{attribute 'linkalways'} 
{attribute 'no_explicit_call' := 'This FB is a CLASS and must be accessed using methods or properties'}
{attribute 'enable_dynamic_creation'}
FUNCTION_BLOCK FINAL EQ_LREAL EXTENDS Node
VAR
	in1 : _LREAL(0.0);
	in2 : _LREAL(0.0);
	out : _BOOL(FALSE);
END_VAR

METHOD PUBLIC Clone : I_Node
VAR
	pNode : POINTER TO EQ_LREAL;
END_VAR
pNode := __NEW(EQ_LREAL);
Clone := pNode^;
END_METHOD

METHOD FB_init : BOOL
VAR_INPUT
	bInitRetains : BOOL; // if TRUE, the retain variables are initialized (warm start / cold start)
	bInCopyCode : BOOL;  // if TRUE, the instance afterwards gets moved into the copy code (online change)
END_VAR
AddInput('in1',THIS^.in1);
AddInput('in2',THIS^.in2);
AddOutput('out', THIS^.out);
END_METHOD

METHOD PROTECTED OnExecute
VAR
END_VAR
out.Value := in1.Value = in2.Value;
END_METHOD

END_FUNCTION_BLOCK

(* stored: Version 1.1.0.1, ProductVersion 3.1.4024.15
   POU EQ_LREAL: Id {bf688540-445c-40be-8eaa-b736cde1f129}, SpecialFunc None
   Folder Constructor: Id {19bb9da7-6860-406a-91fc-f0cf3205dc93}
   Method Clone: Id {9aa511a2-185c-4faf-be91-0902c71d6e26}
   Method FB_init: Id {0c1fef26-acb4-4094-89c9-48de5dc06673}
   Method OnExecute: Id {36fd532a-5121-4432-828c-8893ebf7627d} *)
